_CFC_ (* Continuous Function Chart, elements in execution order *)
#0 AND(NOT SHU6_P2_TS1_DI5, SHU6_P2_KV1_DI8)
#1 TON_Kv1_1:TON(IN: #0, PT: T#10s)
#2 RT_PUSK_OLD:R_TRIG(CLK: #1.Q)
#3 AND(#2.Q, OLD_SOST)
#4 AND(NOT SHU6_P2_TE4_M_ZASCH, SHU6_P2_KV1_DI8)
#5 TON_Kv1_11:TON(IN: #4, PT: T#10s)
#6 RT_PUSK_OLD1:R_TRIG(CLK: #5.Q)
#7 AND(#6.Q, OLD_SOST)
#8 AND(OLD_SOST, SHU6_P2_Z_NET_VH_NAPR)
#9 OR(SHU6_P2_UST_PUSK_VH, #3, #7, #8)
#10 AND(NOT SHU6_P2_UST_RE_OSTANOV, #9)
#11 RT_STOP:R_TRIG(CLK: SHU6_P2_UST_STOP_VH)
#12 OR(#11.Q, SHU6_P2_UST_SET_STOP, SHU6_P2_UST_SET_OSTANOV)
#13 RS_Sost:RS(SET: #10, RESET1: #12)
#14 SHU6_P2_UST_SOST_VKL <= #13.Q1
#15 SHU6_P2_UST_SOST_OTKL <= NOT #13.Q1
#16 AND(NOT SHU6_P2_TS1_DI5, SHU6_P2_KV1_DI8)
#17 TON_Kv11:TON(IN: #16, PT: T#1.5m)
#18 AND(NOT SHU6_P2_TE4_M_ZASCH, SHU6_P2_KV1_DI8)
#19 TON_Kv1:TON(IN: #18, PT: T#1.5m)
#20 AND(#17.Q, #19.Q)
#21 AND(#13.Q1, #20)
#22 AND(NOT #13.Q1, #20)
#23 CTU_TS:CTU(CU: SHU6_P2_TS1_DI5, RESET: #23.Q, PV: 3)
#24 =(#23.CV, 0)
#25 AND(#24, SHU6_P2_TS1_DI5)
#26 TOF_TS_1:TOF(IN: #25, PT: T#60m)
#27 =(#23.CV, 1)
#28 AND(#27, SHU6_P2_TS1_DI5)
#29 TOF_TS_2:TOF(IN: #28, PT: T#60m)
#30 =(#23.CV, 2)
#31 AND(#30, SHU6_P2_TS1_DI5)
#32 TOF_TS_3:TOF(IN: #31, PT: T#60m)
#33 AND(#26.Q, #29.Q, #32.Q)
#34 CTU_Te:CTU(CU: SHU6_P2_TE4_M_ZASCH, RESET: #34.Q, PV: 3)
#35 =(#34.CV, 0)
#36 AND(#35, SHU6_P2_TE4_M_ZASCH)
#37 TOF_TE_1:TOF(IN: #36, PT: T#60m)
#38 =(#34.CV, 1)
#39 AND(#38, SHU6_P2_TE4_M_ZASCH)
#40 TOF_Te_2:TOF(IN: #39, PT: T#60m)
#41 =(#34.CV, 2)
#42 AND(#41, SHU6_P2_TE4_M_ZASCH)
#43 TOF_Te_3:TOF(IN: #42, PT: T#60m)
#44 AND(#37.Q, #40.Q, #43.Q)
#45 OR(#22, #33, #44)
#46 RS_Old_Sost:RS(SET: #21, RESET1: #45)
#47 OLD_SOST <= #46.Q1
_END_CFC_
END_PROGRAM

(* POU Regim/Stop, CFC *)
PROGRAM Stop
VAR
	FT_Ostanov: F_TRIG;
	sr_stop: SR;
	TOF_Progrev: TOF;
END_VAR
VAR (* helpers for the ST form of the networks *)
	_t19 : BOOL;
END_VAR
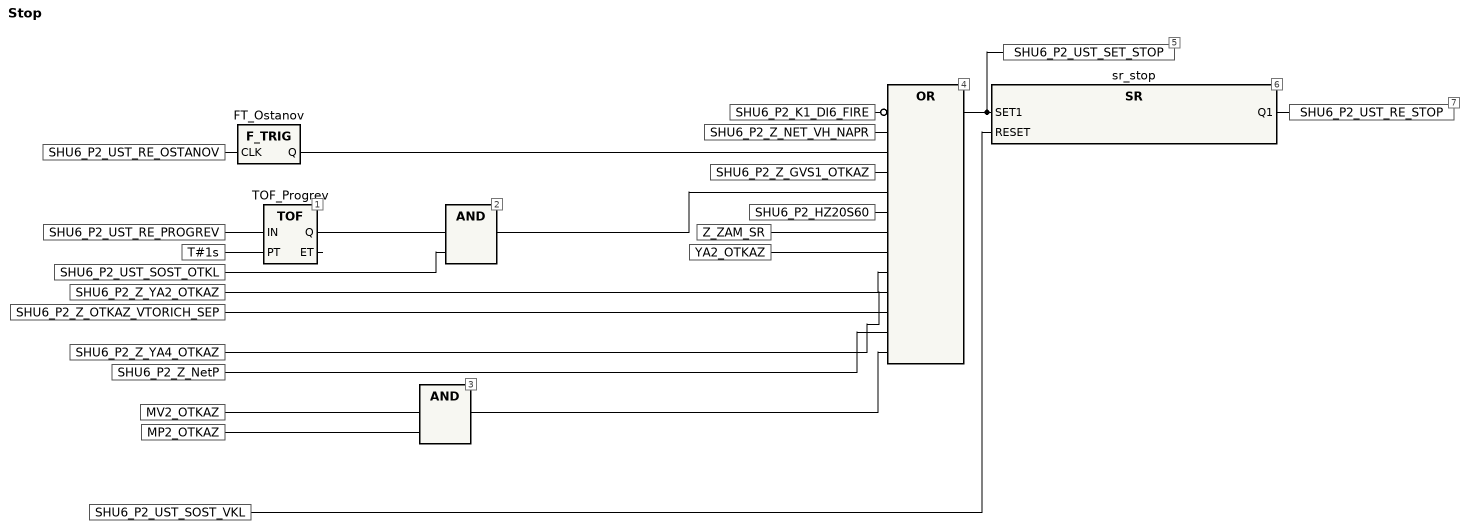
_CFC_ (* Continuous Function Chart, elements in execution order *)
#0 FT_Ostanov:F_TRIG(CLK: SHU6_P2_UST_RE_OSTANOV)
#1 TOF_Progrev:TOF(IN: SHU6_P2_UST_RE_PROGREV, PT: T#1s)
#2 AND(#1.Q, SHU6_P2_UST_SOST_OTKL)
#3 AND(MV2_OTKAZ, MP2_OTKAZ)
#4 OR(NOT SHU6_P2_K1_DI6_FIRE, SHU6_P2_Z_NET_VH_NAPR, #0.Q, SHU6_P2_Z_GVS1_OTKAZ, #2, SHU6_P2_HZ20S60, Z_ZAM_SR, YA2_OTKAZ, SHU6_P2_Z_YA2_OTKAZ, SHU6_P2_Z_OTKAZ_VTORICH_SEP, SHU6_P2_Z_YA4_OTKAZ, SHU6_P2_Z_NetP, #3)
#5 SHU6_P2_UST_SET_STOP <= #4
#6 sr_stop:SR(SET1: #4, RESET: SHU6_P2_UST_SOST_VKL)
#7 SHU6_P2_UST_RE_STOP <= #6.Q1
_END_CFC_
(* the same logic as Structured Text *)
FT_Ostanov(CLK := SHU6_P2_UST_RE_OSTANOV);
TOF_Progrev(IN := SHU6_P2_UST_RE_PROGREV, PT := T#1s);
_t19 := NOT SHU6_P2_K1_DI6_FIRE OR SHU6_P2_Z_NET_VH_NAPR OR FT_Ostanov.Q OR SHU6_P2_Z_GVS1_OTKAZ OR (TOF_Progrev.Q AND SHU6_P2_UST_SOST_OTKL) OR SHU6_P2_HZ20S60 OR Z_ZAM_SR OR YA2_OTKAZ OR SHU6_P2_Z_YA2_OTKAZ OR SHU6_P2_Z_OTKAZ_VTORICH_SEP OR SHU6_P2_Z_YA4_OTKAZ OR SHU6_P2_Z_NetP OR (MV2_OTKAZ AND MP2_OTKAZ);
SHU6_P2_UST_SET_STOP := _t19;
sr_stop(SET1 := _t19, RESET := SHU6_P2_UST_SOST_VKL);
SHU6_P2_UST_RE_STOP := sr_stop.Q1;
END_PROGRAM

(* POU Regim/Ostanov, CFC *)
PROGRAM Ostanov
VAR
	RT_OTKL: R_TRIG;
	SR_OSTANOV: SR;
	TON_AVR_M: TON;
	Z_zam_ostatov: R_TRIG;
END_VAR
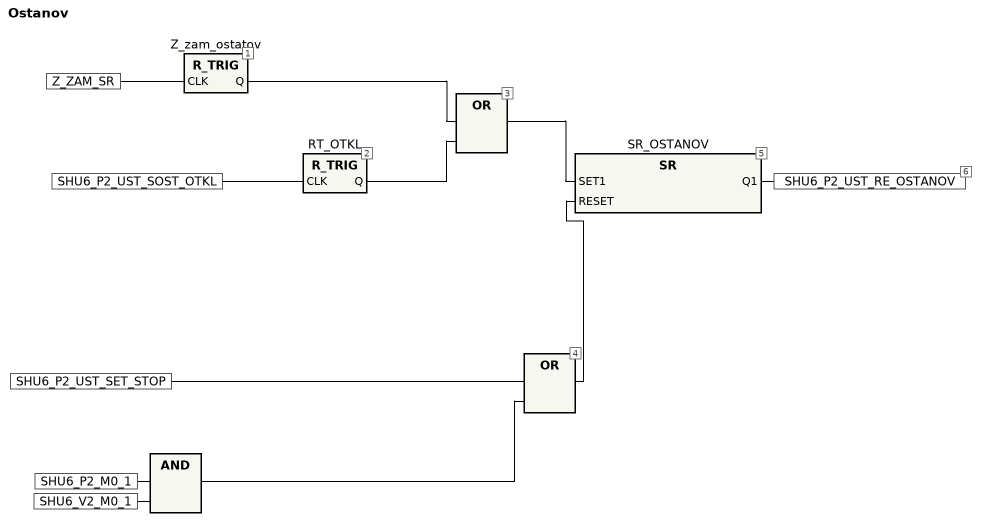
_CFC_ (* Continuous Function Chart, elements in execution order *)
#0 AND(SHU6_P2_M0_1, SHU6_V2_M0_1)
#1 Z_zam_ostatov:R_TRIG(CLK: Z_ZAM_SR)
#2 RT_OTKL:R_TRIG(CLK: SHU6_P2_UST_SOST_OTKL)
#3 OR(#1.Q, #2.Q)
#4 OR(SHU6_P2_UST_SET_STOP, #0)
#5 SR_OSTANOV:SR(SET1: #3, RESET: #4)
#6 SHU6_P2_UST_RE_OSTANOV <= #5.Q1
_END_CFC_
(* the same logic as Structured Text *)
Z_zam_ostatov(CLK := Z_ZAM_SR);
RT_OTKL(CLK := SHU6_P2_UST_SOST_OTKL);
SR_OSTANOV(SET1 := Z_zam_ostatov.Q OR RT_OTKL.Q, RESET := SHU6_P2_UST_SET_STOP OR (SHU6_P2_M0_1 AND SHU6_V2_M0_1));
SHU6_P2_UST_RE_OSTANOV := SR_OSTANOV.Q1;
END_PROGRAM

(* POU Regim/Progrev, CFC *)
PROGRAM Progrev
VAR
	RS_Progrev: RS;
	RT_VKL: R_TRIG;
	TON_SHU6_P2_TE4_M_UST: TON;
	SR_First_On: SR;
END_VAR
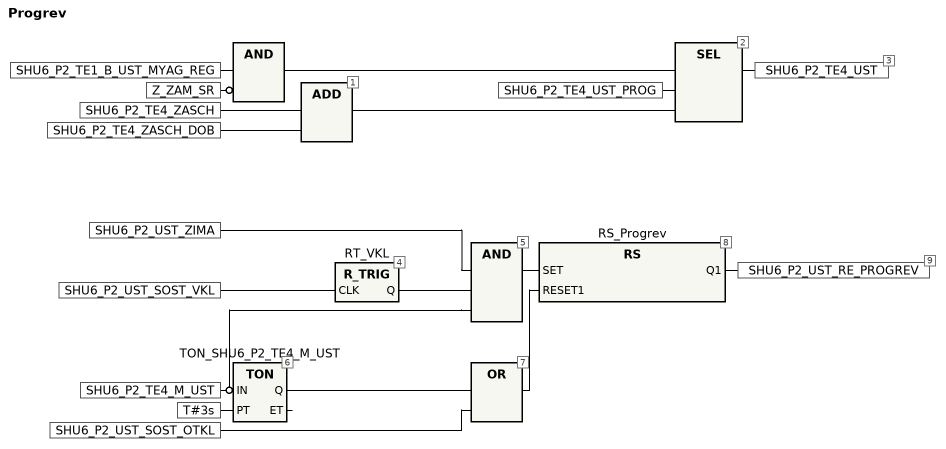
_CFC_ (* Continuous Function Chart, elements in execution order *)
#0 AND(SHU6_P2_TE1_B_UST_MYAG_REG, NOT Z_ZAM_SR)
#1 ADD(SHU6_P2_TE4_ZASCH, SHU6_P2_TE4_ZASCH_DOB)
#2 SEL(#0, SHU6_P2_TE4_UST_PROG, #1)
#3 SHU6_P2_TE4_UST <= #2
#4 RT_VKL:R_TRIG(CLK: SHU6_P2_UST_SOST_VKL)
#5 AND(SHU6_P2_UST_ZIMA, #4.Q, SHU6_P2_TE4_M_UST)
#6 TON_SHU6_P2_TE4_M_UST:TON(IN: NOT SHU6_P2_TE4_M_UST, PT: T#3s)
#7 OR(#6.Q, SHU6_P2_UST_SOST_OTKL)
#8 RS_Progrev:RS(SET: #5, RESET1: #7)
#9 SHU6_P2_UST_RE_PROGREV <= #8.Q1
_END_CFC_
(* the same logic as Structured Text *)
SHU6_P2_TE4_UST := SEL(SHU6_P2_TE1_B_UST_MYAG_REG AND NOT Z_ZAM_SR, SHU6_P2_TE4_UST_PROG, SHU6_P2_TE4_ZASCH + SHU6_P2_TE4_ZASCH_DOB);
RT_VKL(CLK := SHU6_P2_UST_SOST_VKL);
TON_SHU6_P2_TE4_M_UST(IN := NOT SHU6_P2_TE4_M_UST, PT := T#3s);
RS_Progrev(SET := SHU6_P2_UST_ZIMA AND RT_VKL.Q AND SHU6_P2_TE4_M_UST, RESET1 := TON_SHU6_P2_TE4_M_UST.Q OR SHU6_P2_UST_SOST_OTKL);
SHU6_P2_UST_RE_PROGREV := RS_Progrev.Q1;
END_PROGRAM

(* POU Regim/Pusk, CFC *)
PROGRAM Pusk
VAR
	RS_Pusk: RS;
	FT_PROGREV: F_TRIG;
	RT_VKL: R_TRIG;
	TON_sost_VKL: TON;
	TON_AVR_M: TON;
	re_start: F_TRIG;
	TON_Z_ZAM: TON;
END_VAR
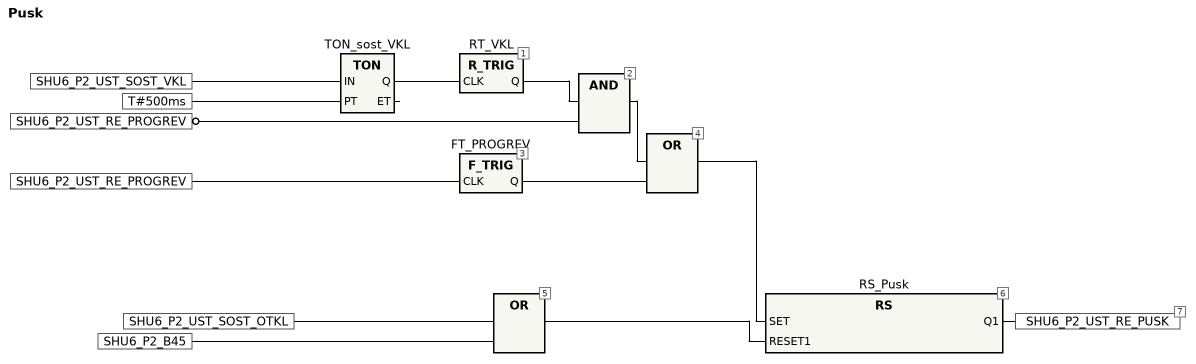
